TYPE ST_Kistler_Status :
STRUCT
	
// =================================================================================
    // KISTLER PRESS HARDWARE STATUS INTERFACE
    // =================================================================================
    bReady       : BOOL :=TRUE; // Hardware is healthy, clear of faults, and ready to press
    bBusy        : BOOL; // Pressing cycle is currently active/running
    bDone        : BOOL; // Cycle completed successfully (Evaluation OK)
    bError       : BOOL; // Press hardware is in a fault condition
    bInPosition  : BOOL; // Press head is at its home/retracted position
	
END_STRUCT
END_TYPE

(* stored: Version 1.1.0.1
   DUT ST_Kistler_Status: Id {13fe1f7e-c843-4ff0-b94a-cef6c7ea4e07} *)
